Fanuc KAREL source: IO0214.KL

PROGRAM IO0214
%NOLOCKGROUP
ROUTINE RTEST
VAR
L1 : ARRAY[3] OF INTEGER;L2 : XYZWPR
L3 : JOINTPOS9
L4 : POSITION
A:BOOLEAN
B:REAL
C:REAL
D:BOOLEAN
E:REAL
BEGIN
--
A=TRUE
L1[1]=2
D=TRUE
E=1.0
L4=$MNUFRAME[1,1]
END RTEST
BEGIN
RTEST
END IO0214
